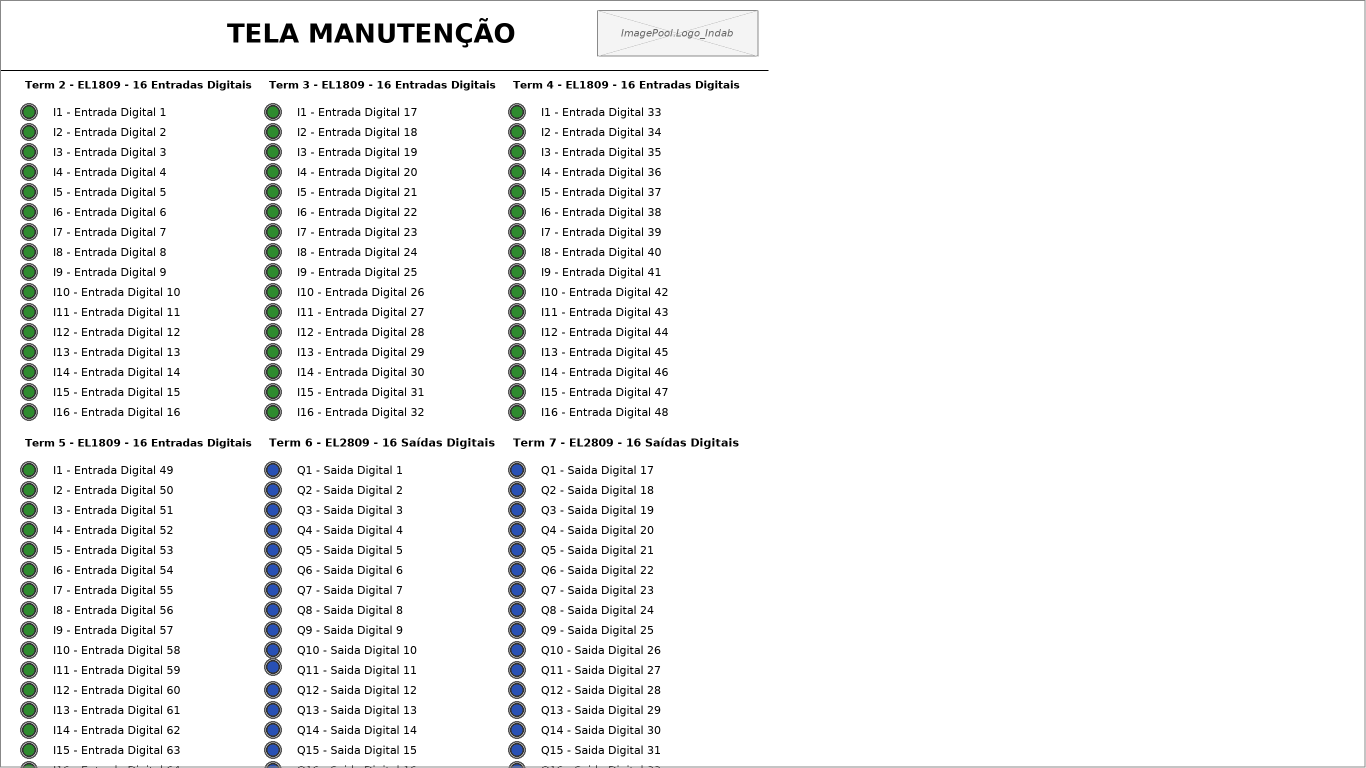
VISUALIZATION Tela_Manutencao  // 1366x768
    Line (0,70) (768,70)
    Line (0,1312) (768,1312)
    Image (597,10 161x46), image: ImagePool.Logo_Indab
    Rectangle (584,1340 180x24), "%t[dd/MM/yyyy]"
    Rectangle (584,1316 180x24), "%t[HH:mm:ss]"
    Label (153,7 437x53), "TELA MANUTENÇÃO"
    Group (19,75 244x347)
        Lamp1 (0,27 20x20), variable: EntradaI0_0, style: Lamp-Lamp1-Green
        Rectangle (31,28 213x19), "I1 - Entrada Digital 1"
        Lamp1 (0,47 20x20), variable: EntradaI0_1, style: Lamp-Lamp1-Green
        Rectangle (31,48 213x19), "I2 - Entrada Digital 2"
        Lamp1 (0,67 20x20), variable: EntradaI0_2, style: Lamp-Lamp1-Green
        Rectangle (31,68 213x19), "I3 - Entrada Digital 3"
        Lamp1 (0,87 20x20), variable: EntradaI0_3, style: Lamp-Lamp1-Green
        Rectangle (31,88 213x19), "I4 - Entrada Digital 4"
        Lamp1 (0,107 20x20), variable: EntradaI0_4, style: Lamp-Lamp1-Green
        Rectangle (31,108 213x19), "I5 - Entrada Digital 5"
        Lamp1 (0,127 20x20), variable: EntradaI0_5, style: Lamp-Lamp1-Green
        Rectangle (31,128 213x19), "I6 - Entrada Digital 6"
        Lamp1 (0,147 20x20), variable: EntradaI0_6, style: Lamp-Lamp1-Green
        Rectangle (31,148 213x19), "I7 - Entrada Digital 7"
        Lamp1 (0,167 20x20), variable: EntradaI0_7, style: Lamp-Lamp1-Green
        Rectangle (31,168 213x19), "I8 - Entrada Digital 8"
        Lamp1 (0,187 20x20), variable: EntradaI1_0, style: Lamp-Lamp1-Green
        Rectangle (31,188 213x19), "I9 - Entrada Digital 9"
        Lamp1 (0,207 20x20), variable: EntradaI1_1, style: Lamp-Lamp1-Green
        Rectangle (31,208 213x19), "I10 - Entrada Digital 10"
        Lamp1 (0,227 20x20), variable: EntradaI1_2, style: Lamp-Lamp1-Green
        Rectangle (31,228 213x19), "I11 - Entrada Digital 11"
        Lamp1 (0,247 20x20), variable: EntradaI1_3, style: Lamp-Lamp1-Green
        Rectangle (31,248 213x19), "I12 - Entrada Digital 12"
        Lamp1 (0,267 20x20), variable: EntradaI1_4, style: Lamp-Lamp1-Green
        Rectangle (31,268 213x19), "I13 - Entrada Digital 13"
        Lamp1 (0,287 20x20), variable: EntradaI1_5, style: Lamp-Lamp1-Green
        Rectangle (31,288 213x19), "I14 - Entrada Digital 14"
        Lamp1 (0,307 20x20), variable: EntradaI1_6, style: Lamp-Lamp1-Green
        Rectangle (31,308 213x19), "I15 - Entrada Digital 15"
        Lamp1 (0,327 20x20), variable: EntradaI1_7, style: Lamp-Lamp1-Green
        Rectangle (31,328 213x19), "I16 - Entrada Digital 16"
        Rectangle (3,0 237x20), "Term 2 - EL1809 - 16 Entradas Digitais"
    Group (19,433 244x347)
        Lamp1 (0,27 20x20), variable: EntradaI6_0, style: Lamp-Lamp1-Green
        Rectangle (31,28 213x19), "I1 - Entrada Digital 49"
        Lamp1 (0,47 20x20), variable: EntradaI6_1, style: Lamp-Lamp1-Green
        Rectangle (31,48 213x19), "I2 - Entrada Digital 50"
        Lamp1 (0,67 20x20), variable: EntradaI6_2, style: Lamp-Lamp1-Green
        Rectangle (31,68 213x19), "I3 - Entrada Digital 51"
        Lamp1 (0,87 20x20), variable: EntradaI6_3, style: Lamp-Lamp1-Green
        Rectangle (31,88 213x19), "I4 - Entrada Digital 52"
        Lamp1 (0,107 20x20), variable: EntradaI6_4, style: Lamp-Lamp1-Green
        Rectangle (31,108 213x19), "I5 - Entrada Digital 53"
        Lamp1 (0,127 20x20), variable: EntradaI6_5, style: Lamp-Lamp1-Green
        Rectangle (31,128 213x19), "I6 - Entrada Digital 54"
        Lamp1 (0,147 20x20), variable: EntradaI6_6, style: Lamp-Lamp1-Green
        Rectangle (31,148 213x19), "I7 - Entrada Digital 55"
        Lamp1 (0,167 20x20), variable: EntradaI6_7, style: Lamp-Lamp1-Green
        Rectangle (31,168 213x19), "I8 - Entrada Digital 56"
        Lamp1 (0,187 20x20), variable: EntradaI7_0, style: Lamp-Lamp1-Green
        Rectangle (31,188 213x19), "I9 - Entrada Digital 57"
        Lamp1 (0,207 20x20), variable: EntradaI7_1, style: Lamp-Lamp1-Green
        Rectangle (31,208 213x19), "I10 - Entrada Digital 58"
        Lamp1 (0,227 20x20), variable: EntradaI7_2, style: Lamp-Lamp1-Green
        Rectangle (31,228 213x19), "I11 - Entrada Digital 59"
        Lamp1 (0,247 20x20), variable: EntradaI7_3, style: Lamp-Lamp1-Green
        Rectangle (31,248 213x19), "I12 - Entrada Digital 60"
        Lamp1 (0,267 20x20), variable: EntradaI7_4, style: Lamp-Lamp1-Green
        Rectangle (31,268 213x19), "I13 - Entrada Digital 61"
        Lamp1 (0,287 20x20), variable: EntradaI7_5, style: Lamp-Lamp1-Green
        Rectangle (31,288 213x19), "I14 - Entrada Digital 62"
        Lamp1 (0,307 20x20), variable: EntradaI7_6, style: Lamp-Lamp1-Green
        Rectangle (31,308 213x19), "I15 - Entrada Digital 63"
        Lamp1 (0,327 20x20), variable: EntradaI7_7, style: Lamp-Lamp1-Green
        Rectangle (31,328 213x19), "I16 - Entrada Digital 64"
        Rectangle (3,0 237x20), "Term 5 - EL1809 - 16 Entradas Digitais"
    Group (263,75 244x347)
        Lamp1 (0,27 20x20), variable: EntradaI2_0, style: Lamp-Lamp1-Green
        Rectangle (31,28 213x19), "I1 - Entrada Digital 17"
        Lamp1 (0,47 20x20), variable: EntradaI2_1, style: Lamp-Lamp1-Green
        Rectangle (31,48 213x19), "I2 - Entrada Digital 18"
        Lamp1 (0,67 20x20), variable: EntradaI2_2, style: Lamp-Lamp1-Green
        Rectangle (31,68 213x19), "I3 - Entrada Digital 19"
        Lamp1 (0,87 20x20), variable: EntradaI2_3, style: Lamp-Lamp1-Green
        Rectangle (31,88 213x19), "I4 - Entrada Digital 20"
        Lamp1 (0,107 20x20), variable: EntradaI2_4, style: Lamp-Lamp1-Green
        Rectangle (31,108 213x19), "I5 - Entrada Digital 21"
        Lamp1 (0,127 20x20), variable: EntradaI2_5, style: Lamp-Lamp1-Green
        Rectangle (31,128 213x19), "I6 - Entrada Digital 22"
        Lamp1 (0,147 20x20), variable: EntradaI2_6, style: Lamp-Lamp1-Green
        Rectangle (31,148 213x19), "I7 - Entrada Digital 23"
        Lamp1 (0,167 20x20), variable: EntradaI2_7, style: Lamp-Lamp1-Green
        Rectangle (31,168 213x19), "I8 - Entrada Digital 24"
        Lamp1 (0,187 20x20), variable: EntradaI3_0, style: Lamp-Lamp1-Green
        Rectangle (31,188 213x19), "I9 - Entrada Digital 25"
        Lamp1 (0,207 20x20), variable: EntradaI3_1, style: Lamp-Lamp1-Green
        Rectangle (31,208 213x19), "I10 - Entrada Digital 26"
        Lamp1 (0,227 20x20), variable: EntradaI3_2, style: Lamp-Lamp1-Green
        Rectangle (31,228 213x19), "I11 - Entrada Digital 27"
        Lamp1 (0,247 20x20), variable: EntradaI3_3, style: Lamp-Lamp1-Green
        Rectangle (31,248 213x19), "I12 - Entrada Digital 28"
        Lamp1 (0,267 20x20), variable: EntradaI3_4, style: Lamp-Lamp1-Green
        Rectangle (31,268 213x19), "I13 - Entrada Digital 29"
        Lamp1 (0,287 20x20), variable: EntradaI3_5, style: Lamp-Lamp1-Green
        Rectangle (31,288 213x19), "I14 - Entrada Digital 30"
        Lamp1 (0,307 20x20), variable: EntradaI3_6, style: Lamp-Lamp1-Green
        Rectangle (31,308 213x19), "I15 - Entrada Digital 31"
        Lamp1 (0,327 20x20), variable: EntradaI3_7, style: Lamp-Lamp1-Green
        Rectangle (31,328 213x19), "I16 - Entrada Digital 32"
        Rectangle (3,0 239x20), "Term 3 - EL1809 - 16 Entradas Digitais"
    Group (507,75 244x347)
        Lamp1 (0,27 20x20), variable: EntradaI4_0, style: Lamp-Lamp1-Green
        Rectangle (31,28 213x19), "I1 - Entrada Digital 33"
        Lamp1 (0,47 20x20), variable: EntradaI4_1, style: Lamp-Lamp1-Green
        Rectangle (31,48 213x19), "I2 - Entrada Digital 34"
        Lamp1 (0,67 20x20), variable: EntradaI4_2, style: Lamp-Lamp1-Green
        Rectangle (31,68 213x19), "I3 - Entrada Digital 35"
        Lamp1 (0,87 20x20), variable: EntradaI4_3, style: Lamp-Lamp1-Green
        Rectangle (31,88 213x19), "I4 - Entrada Digital 36"
        Lamp1 (0,107 20x20), variable: EntradaI4_4, style: Lamp-Lamp1-Green
        Rectangle (31,108 213x19), "I5 - Entrada Digital 37"
        Lamp1 (0,127 20x20), variable: EntradaI4_5, style: Lamp-Lamp1-Green
        Rectangle (31,128 213x19), "I6 - Entrada Digital 38"
        Lamp1 (0,147 20x20), variable: EntradaI4_6, style: Lamp-Lamp1-Green
        Rectangle (31,148 213x19), "I7 - Entrada Digital 39"
        Lamp1 (0,167 20x20), variable: EntradaI4_7, style: Lamp-Lamp1-Green
        Rectangle (31,168 213x19), "I8 - Entrada Digital 40"
        Lamp1 (0,187 20x20), variable: EntradaI5_0, style: Lamp-Lamp1-Green
        Rectangle (31,188 213x19), "I9 - Entrada Digital 41"
        Lamp1 (0,207 20x20), variable: EntradaI5_1, style: Lamp-Lamp1-Green
        Rectangle (31,208 213x19), "I10 - Entrada Digital 42"
        Lamp1 (0,227 20x20), variable: EntradaI5_2, style: Lamp-Lamp1-Green
        Rectangle (31,228 213x19), "I11 - Entrada Digital 43"
        Lamp1 (0,247 20x20), variable: EntradaI5_3, style: Lamp-Lamp1-Green
        Rectangle (31,248 213x19), "I12 - Entrada Digital 44"
        Lamp1 (0,267 20x20), variable: EntradaI5_4, style: Lamp-Lamp1-Green
        Rectangle (31,268 213x19), "I13 - Entrada Digital 45"
        Lamp1 (0,287 20x20), variable: EntradaI5_5, style: Lamp-Lamp1-Green
        Rectangle (31,288 213x19), "I14 - Entrada Digital 46"
        Lamp1 (0,307 20x20), variable: EntradaI5_6, style: Lamp-Lamp1-Green
        Rectangle (31,308 213x19), "I15 - Entrada Digital 47"
        Lamp1 (0,327 20x20), variable: EntradaI5_7, style: Lamp-Lamp1-Green
        Rectangle (31,328 213x19), "I16 - Entrada Digital 48"
        Rectangle (3,0 237x20), "Term 4 - EL1809 - 16 Entradas Digitais"
    Group (263,433 244x347)
        Lamp1 (0,27 20x20), variable: SaidaQ0_0, style: Lamp-Lamp1-Blue
        Rectangle (31,28 213x19), "Q1 - Saida Digital 1"
        Lamp1 (0,47 20x20), variable: SaidaQ0_1, style: Lamp-Lamp1-Blue
        Rectangle (31,48 213x19), "Q2 - Saida Digital 2"
        Lamp1 (0,67 20x20), variable: SaidaQ0_2, style: Lamp-Lamp1-Blue
        Rectangle (31,68 213x19), "Q3 - Saida Digital 3"
        Lamp1 (0,87 20x20), variable: SaidaQ0_3, style: Lamp-Lamp1-Blue
        Rectangle (31,88 213x19), "Q4 - Saida Digital 4"
        Lamp1 (0,107 20x20), variable: SaidaQ0_4, style: Lamp-Lamp1-Blue
        Rectangle (31,108 213x19), "Q5 - Saida Digital 5"
        Lamp1 (0,127 20x20), variable: SaidaQ0_5, style: Lamp-Lamp1-Blue
        Rectangle (31,128 213x19), "Q6 - Saida Digital 6"
        Lamp1 (0,147 20x20), variable: SaidaQ0_6, style: Lamp-Lamp1-Blue
        Rectangle (31,148 213x19), "Q7 - Saida Digital 7"
        Lamp1 (0,167 20x20), variable: SaidaQ0_7, style: Lamp-Lamp1-Blue
        Rectangle (31,168 213x19), "Q8 - Saida Digital 8"
        Lamp1 (0,187 20x20), variable: SaidaQ1_0, style: Lamp-Lamp1-Blue
        Rectangle (31,188 213x19), "Q9 - Saida Digital 9"
        Lamp1 (0,207 20x20), variable: SaidaQ1_1, style: Lamp-Lamp1-Blue
        Rectangle (31,208 213x19), "Q10 - Saida Digital 10"
        Lamp1 (0,224 20x20), variable: SaidaQ1_2, style: Lamp-Lamp1-Blue
        Rectangle (31,228 213x19), "Q11 - Saida Digital 11"
        Lamp1 (0,247 20x20), variable: SaidaQ1_3, style: Lamp-Lamp1-Blue
        Rectangle (31,248 213x19), "Q12 - Saida Digital 12"
        Lamp1 (0,267 20x20), variable: SaidaQ1_4, style: Lamp-Lamp1-Blue
        Rectangle (31,268 213x19), "Q13 - Saida Digital 13"
        Lamp1 (0,287 20x20), variable: SaidaQ1_5, style: Lamp-Lamp1-Blue
        Rectangle (31,288 213x19), "Q14 - Saida Digital 14"
        Lamp1 (0,307 20x20), variable: SaidaQ1_6, style: Lamp-Lamp1-Blue
        Rectangle (31,308 213x19), "Q15 - Saida Digital 15"
        Lamp1 (0,327 20x20), variable: SaidaQ1_7, style: Lamp-Lamp1-Blue
        Rectangle (31,328 213x19), "Q16 - Saida Digital 16"
        Rectangle (3,0 237x20), "Term 6 - EL2809 - 16 Saídas Digitais"
    Group (507,433 244x347)
        Lamp1 (0,27 20x20), variable: SaidaQ2_0, style: Lamp-Lamp1-Blue
        Rectangle (31,28 213x19), "Q1 - Saida Digital 17"
        Lamp1 (0,47 20x20), variable: SaidaQ2_1, style: Lamp-Lamp1-Blue
        Rectangle (31,48 213x19), "Q2 - Saida Digital 18"
        Lamp1 (0,67 20x20), variable: SaidaQ2_2, style: Lamp-Lamp1-Blue
        Rectangle (31,68 213x19), "Q3 - Saida Digital 19"
        Lamp1 (0,87 20x20), variable: SaidaQ2_3, style: Lamp-Lamp1-Blue
        Rectangle (31,88 213x19), "Q4 - Saida Digital 20"
        Lamp1 (0,107 20x20), variable: SaidaQ2_4, style: Lamp-Lamp1-Blue
        Rectangle (31,108 213x19), "Q5 - Saida Digital 21"
        Lamp1 (0,127 20x20), variable: SaidaQ2_5, style: Lamp-Lamp1-Blue
        Rectangle (31,128 213x19), "Q6 - Saida Digital 22"
        Lamp1 (0,147 20x20), variable: SaidaQ2_6, style: Lamp-Lamp1-Blue
        Rectangle (31,148 213x19), "Q7 - Saida Digital 23"
        Lamp1 (0,167 20x20), variable: SaidaQ2_7, style: Lamp-Lamp1-Blue
        Rectangle (31,168 213x19), "Q8 - Saida Digital 24"
        Lamp1 (0,187 20x20), variable: SaidaQ3_0, style: Lamp-Lamp1-Blue
        Rectangle (31,188 213x19), "Q9 - Saida Digital 25"
        Lamp1 (0,207 20x20), variable: SaidaQ3_1, style: Lamp-Lamp1-Blue
        Rectangle (31,208 213x19), "Q10 - Saida Digital 26"
        Lamp1 (0,227 20x20), variable: SaidaQ3_2, style: Lamp-Lamp1-Blue
        Rectangle (31,228 213x19), "Q11 - Saida Digital 27"
        Lamp1 (0,247 20x20), variable: SaidaQ3_3, style: Lamp-Lamp1-Blue
        Rectangle (31,248 213x19), "Q12 - Saida Digital 28"
        Lamp1 (0,267 20x20), variable: SaidaQ3_4, style: Lamp-Lamp1-Blue
        Rectangle (31,268 213x19), "Q13 - Saida Digital 29"
        Lamp1 (0,287 20x20), variable: SaidaQ3_5, style: Lamp-Lamp1-Blue
        Rectangle (31,288 213x19), "Q14 - Saida Digital 30"
        Lamp1 (0,307 20x20), variable: SaidaQ3_6, style: Lamp-Lamp1-Blue
        Rectangle (31,308 213x19), "Q15 - Saida Digital 31"
        Lamp1 (0,327 20x20), variable: SaidaQ3_7, style: Lamp-Lamp1-Blue
        Rectangle (31,328 213x19), "Q16 - Saida Digital 32"
        Rectangle (3,0 237x20), "Term 7 - EL2809 - 16 Saídas Digitais"
    Group (19,791 244x347)
        Lamp1 (0,27 20x20), variable: SaidaQ4_0, style: Lamp-Lamp1-Blue
        Rectangle (31,28 213x19), "Q1 - Saida Digital 33"
        Lamp1 (0,47 20x20), variable: SaidaQ4_1, style: Lamp-Lamp1-Blue
        Rectangle (31,48 213x19), "Q2 - Saida Digital 34"
        Lamp1 (0,67 20x20), variable: SaidaQ4_2, style: Lamp-Lamp1-Blue
        Rectangle (31,68 213x19), "Q3 - Saida Digital 35"
        Lamp1 (0,87 20x20), variable: SaidaQ4_3, style: Lamp-Lamp1-Blue
        Rectangle (31,88 213x19), "Q4 - Saida Digital 36"
        Lamp1 (0,107 20x20), variable: SaidaQ4_4, style: Lamp-Lamp1-Blue
        Rectangle (31,108 213x19), "Q5 - Saida Digital 37"
        Lamp1 (0,127 20x20), variable: SaidaQ4_5, style: Lamp-Lamp1-Blue
        Rectangle (31,128 213x19), "Q6 - Saida Digital 38"
        Lamp1 (0,147 20x20), variable: SaidaQ4_6, style: Lamp-Lamp1-Blue
        Rectangle (31,148 213x19), "Q7 - Saida Digital 39"
        Lamp1 (0,167 20x20), variable: SaidaQ4_7, style: Lamp-Lamp1-Blue
        Rectangle (31,168 213x19), "Q8 - Saida Digital 40"
        Lamp1 (0,187 20x20), variable: SaidaQ5_0, style: Lamp-Lamp1-Blue
        Rectangle (31,188 213x19), "Q9 - Saida Digital 41"
        Lamp1 (0,207 20x20), variable: SaidaQ5_1, style: Lamp-Lamp1-Blue
        Rectangle (31,208 213x19), "Q10 - Saida Digital 42"
        Lamp1 (0,227 20x20), variable: SaidaQ5_2, style: Lamp-Lamp1-Blue
        Rectangle (31,228 213x19), "Q11 - Saida Digital 43"
        Lamp1 (0,247 20x20), variable: SaidaQ5_3, style: Lamp-Lamp1-Blue
        Rectangle (31,248 213x19), "Q12 - Saida Digital 44"
        Lamp1 (0,267 20x20), variable: SaidaQ5_4, style: Lamp-Lamp1-Blue
        Rectangle (31,268 213x19), "Q13 - Saida Digital 45"
        Lamp1 (0,287 20x20), variable: SaidaQ5_5, style: Lamp-Lamp1-Blue
        Rectangle (31,288 213x19), "Q14 - Saida Digital 46"
        Lamp1 (0,307 20x20), variable: SaidaQ5_6, style: Lamp-Lamp1-Blue
        Rectangle (31,308 213x19), "Q15 - Saida Digital 47"
        Lamp1 (0,327 20x20), variable: SaidaQ5_7, style: Lamp-Lamp1-Blue
        Rectangle (31,328 213x19), "Q16 - Saida Digital 48"
        Rectangle (3,0 237x20), "Term 8 - EL2809 - 16 Saídas Digitais"
    Group (263,791 244x347)
        Lamp1 (0,27 20x20), variable: SaidaQ6_0, style: Lamp-Lamp1-Blue
        Rectangle (31,28 213x19), "Q1 - Saida Digital 49"
        Lamp1 (0,47 20x20), variable: SaidaQ6_1, style: Lamp-Lamp1-Blue
        Rectangle (31,48 213x19), "Q2 - Saida Digital 50"
        Lamp1 (0,67 20x20), variable: SaidaQ6_2, style: Lamp-Lamp1-Blue
        Rectangle (31,68 213x19), "Q3 - Saida Digital 51"
        Lamp1 (0,87 20x20), variable: SaidaQ6_3, style: Lamp-Lamp1-Blue
        Rectangle (31,88 213x19), "Q4 - Saida Digital 52"
        Lamp1 (0,107 20x20), variable: SaidaQ6_4, style: Lamp-Lamp1-Blue
        Rectangle (31,108 213x19), "Q5 - Saida Digital 53"
        Lamp1 (0,127 20x20), variable: SaidaQ6_5, style: Lamp-Lamp1-Blue
        Rectangle (31,128 213x19), "Q6 - Saida Digital 54"
        Lamp1 (0,147 20x20), variable: SaidaQ6_7, style: Lamp-Lamp1-Blue
        Rectangle (31,148 213x19), "Q7 - Saida Digital 55"
        Lamp1 (0,167 20x20), variable: SaidaQ7_0, style: Lamp-Lamp1-Blue
        Rectangle (31,168 213x19), "Q8 - Saida Digital 56"
        Lamp1 (0,187 20x20), variable: SaidaQ7_1, style: Lamp-Lamp1-Blue
        Rectangle (31,188 213x19), "Q9 - Saida Digital 57"
        Lamp1 (0,207 20x20), variable: SaidaQ7_1, style: Lamp-Lamp1-Blue
        Rectangle (31,208 213x19), "Q10 - Saida Digital 58"
        Lamp1 (0,227 20x20), variable: SaidaQ7_2, style: Lamp-Lamp1-Blue
        Rectangle (31,228 213x19), "Q11 - Saida Digital 59"
        Lamp1 (0,247 20x20), variable: SaidaQ7_3, style: Lamp-Lamp1-Blue
        Rectangle (31,248 213x19), "Q12 - Saida Digital 60"
        Lamp1 (0,267 20x20), variable: SaidaQ7_4, style: Lamp-Lamp1-Blue
        Rectangle (31,268 213x19), "Q13 - Saida Digital 61"
        Lamp1 (0,287 20x20), variable: SaidaQ7_5, style: Lamp-Lamp1-Blue
        Rectangle (31,288 213x19), "Q14 - Saida Digital 62"
        Lamp1 (0,307 20x20), variable: SaidaQ7_6, style: Lamp-Lamp1-Blue
        Rectangle (31,308 213x19), "Q15 - Saida Digital 63"
        Lamp1 (0,327 20x20), variable: SaidaQ7_7, style: Lamp-Lamp1-Blue
        Rectangle (31,328 213x19), "Q16 - Saida Digital 64"
        Rectangle (3,0 237x20), "Term 9 - EL2809 - 16 Saídas Digitais"
    Group (263,1242 244x67)
        Lamp1 (0,27 20x20), variable: I2, style: Lamp-Lamp1-Yellow
        Rectangle (31,28 213x19), "I1 - Entrada Rapida 1"
        Lamp1 (0,47 20x20), variable: I2, style: Lamp-Lamp1-Yellow
        Rectangle (31,48 213x19), "I2 - Entrada Rapida 2"
        Rectangle (3,0 237x20), "Term 9 - EL1252 - 2 Entradas Rápidas"
    Group (19,1146 244x104)
        Rectangle (0,0 237x20), "Term 9 - EL4004 - 4 Saídas Analógicas"
        Group (51,28 202x76)
            Rectangle (0,0 213x19), "AO1 - Saida Analogica 1"
            Rectangle (0,19 213x19), "AO1 - Saida Analogica 2"
            Rectangle (0,38 213x19), "AO1 - Saida Analogica 3"
            Rectangle (0,57 213x19), "AO1 - Saida Analogica 4"
        Group (0,28 51x76)
            Rectangle (0,0 51x19), "%s"
            Rectangle (0,19 51x19), "%s"
            Rectangle (0,38 51x19), "%s"
            Rectangle (0,57 51x19), "%s"
    Group (263,1146 244x87)
        Lamp1 (0,27 20x20), variable: I2, style: Lamp-Lamp1-Yellow
        Rectangle (31,28 213x19), "Robo Yaskawa GP7"
        Lamp1 (0,47 20x20), variable: I2, style: Lamp-Lamp1-Yellow
        Rectangle (31,48 213x19), "Camera Sick Inspector"
        Rectangle (3,0 237x20), "Conexão Ethernet/IP"
        Lamp1 (0,67 20x20), variable: I2, style: Lamp-Lamp1-Yellow
        Rectangle (31,68 213x19), "Safety Sick Flexi Soft"
    Rectangle (510,791 237x20), "Dispositivos Safety"
    Rectangle (510,809 237x20), "XTIO[1] - 8 entradas e 4 Saídas"
    Rectangle (547,829 204x19), "I1-I2 - Botão de Emergência"
    Lamp1 (507,829 20x20), variable: I2, style: Lamp-Lamp1-Yellow
    Lamp1 (527,829 20x20), variable: I2, style: Lamp-Lamp1-Yellow
    Rectangle (547,849 204x19), "I3-I4 - Botão de Emergência"
    Lamp1 (507,849 20x20), variable: I2, style: Lamp-Lamp1-Yellow
    Lamp1 (527,849 20x20), variable: I2, style: Lamp-Lamp1-Yellow
    Lamp1 (507,869 20x20), variable: I2, style: Lamp-Lamp1-Yellow
    Rectangle (547,869 204x19), "I3-I4 - Botão de Emergência"
    Lamp1 (527,869 20x20), variable: I2, style: Lamp-Lamp1-Yellow
    Lamp1 (507,889 20x20), variable: I2, style: Lamp-Lamp1-Yellow
    Rectangle (547,889 204x19), "I3-I4 - Botão de Emergência"
    Lamp1 (527,889 20x20), variable: I2, style: Lamp-Lamp1-Yellow
    Lamp1 (507,909 20x20), variable: I2, style: Lamp-Lamp1-Yellow
    Rectangle (547,909 204x19), "Q1-Q2 - Servo 1"
    Lamp1 (527,909 20x20), variable: I2, style: Lamp-Lamp1-Yellow
    Lamp1 (507,929 20x20), variable: I2, style: Lamp-Lamp1-Yellow
    Rectangle (547,929 204x19), "Q3-Q4 - Servo 2"
    Lamp1 (527,929 20x20), variable: I2, style: Lamp-Lamp1-Yellow
    Rectangle (510,952 237x20), "XTIO[2] - 8 entradas e 4 Saídas"
    Rectangle (547,972 204x19), "I1-I2 - Cortina de Luz"
    Lamp1 (507,972 20x20), variable: I2, style: Lamp-Lamp1-Yellow
    Lamp1 (527,972 20x20), variable: I2, style: Lamp-Lamp1-Yellow
    Rectangle (547,992 204x19), "I3-I4 - Sensor Porta"
    Lamp1 (507,992 20x20), variable: I2, style: Lamp-Lamp1-Yellow
    Lamp1 (527,992 20x20), variable: I2, style: Lamp-Lamp1-Yellow
    Lamp1 (507,1012 20x20), variable: I2, style: Lamp-Lamp1-Yellow
    Rectangle (547,1012 204x19), "I3-I4 - Sensor Porta"
    Lamp1 (527,1012 20x20), variable: I2, style: Lamp-Lamp1-Yellow
    Lamp1 (507,1032 20x20), variable: I2, style: Lamp-Lamp1-Yellow
    Rectangle (547,1032 204x19), "I3-I4 - Sensor Porta"
    Lamp1 (527,1032 20x20), variable: I2, style: Lamp-Lamp1-Yellow
    Lamp1 (507,1052 20x20), variable: I2, style: Lamp-Lamp1-Yellow
    Rectangle (547,1052 204x19), "Q1-Q2 - Motor"
    Lamp1 (527,1052 20x20), variable: I2, style: Lamp-Lamp1-Yellow
    Lamp1 (507,1072 20x20), variable: I2, style: Lamp-Lamp1-Yellow
    Rectangle (547,1072 204x19), "Q3-Q4 - Motor"
    Lamp1 (527,1072 20x20), variable: I2, style: Lamp-Lamp1-Yellow
    Rectangle (507,1094 237x20), "XTIO[3] - 8 entradas e 4 Saídas"
    Rectangle (544,1114 204x19), "I1-I2 - Sensor Porta"
    Lamp1 (504,1114 20x20), variable: I2, style: Lamp-Lamp1-Yellow
    Lamp1 (524,1114 20x20), variable: I2, style: Lamp-Lamp1-Yellow
    Rectangle (544,1134 204x19), "I3-I4 - Sensor Porta"
    Lamp1 (504,1134 20x20), variable: I2, style: Lamp-Lamp1-Yellow
    Lamp1 (524,1134 20x20), variable: I2, style: Lamp-Lamp1-Yellow
    Lamp1 (504,1154 20x20), variable: I2, style: Lamp-Lamp1-Yellow
    Rectangle (544,1154 204x19), "I3-I4 - Sensor Porta"
    Lamp1 (524,1154 20x20), variable: I2, style: Lamp-Lamp1-Yellow
    Lamp1 (504,1174 20x20), variable: I2, style: Lamp-Lamp1-Yellow
    Rectangle (544,1174 204x19), "I3-I4 - Sensor Porta"
    Lamp1 (524,1174 20x20), variable: I2, style: Lamp-Lamp1-Yellow
    Lamp1 (504,1194 20x20), variable: I2, style: Lamp-Lamp1-Yellow
    Rectangle (544,1194 204x19), "Q1-Q2 - Robo Yaskawa GP7"
    Lamp1 (524,1194 20x20), variable: I2, style: Lamp-Lamp1-Yellow
    Lamp1 (504,1214 20x20), variable: I2, style: Lamp-Lamp1-Yellow
    Rectangle (544,1214 204x19), "Q3-Q4 - Reserva"
    Lamp1 (524,1214 20x20), variable: I2, style: Lamp-Lamp1-Yellow
    Button (15,1315 175x45), "RECEITAS"
        OnMouseClick: change screen: Tela_Receita
    Button (375,1315 175x45), "MOV. MANUAIS"
        OnMouseClick: change screen: Tela_Manual_1
    Button (195,1315 175x45), "PRODUÇÃO"
        OnMouseClick: change screen: Tela_Producao
END_VISUALIZATION

(* stored: Version 1.1.0.1, ProductVersion 3.1.4024.11
   Visu Tela_Manutencao: Id {edb76721-bd18-451d-ba38-75c6ea792aa9} *)
